# EPICS substitutions: iocCollimatorControl/R27CLM.substitutions
#BO,EPICS->PLC,Command
file "../../db/bo_word.template"{ pattern
{	P,		R,					PORT,		OFFSET,		MASK,		ZNAM,		ONAM	}
{	SR:R27:CLM:R27CLM:,	btn_LocalOrRemote,			R27CLM_BO1_Bits,	0,		0x0001,		Low,		High	}
{	SR:R27:CLM:R27CLM:,	btn_E_STOP,				R27CLM_BO1_Bits,	0,		0x0002,		Low,		High	}
{	SR:R27:CLM:R27CLM:,	m_restartTC,				R27CLM_BO1_Bits,	0,		0x0004,		Low,		High	}
{	SR:R27:CLM:R27CLM:,	btn_Move_Axis1,				R27CLM_BO2_Bits,	0,		0x0001,		Low,		High	}
{	SR:R27:CLM:R27CLM:,	btn_JogForward_Axis1,			R27CLM_BO2_Bits,	0,		0x0002,		Low,		High	}
{	SR:R27:CLM:R27CLM:,	btn_JogBackward_Axis1,			R27CLM_BO2_Bits,	0,		0x0004,		Low,		High	}
{	SR:R27:CLM:R27CLM:,	btn_Stop_Axis1,				R27CLM_BO2_Bits,	0,		0x0008,		Low,		High	}
{	SR:R27:CLM:R27CLM:,	btn_Reset_Axis1,			R27CLM_BO2_Bits,	0,		0x0010,		Low,		High	}
{	SR:R27:CLM:R27CLM:,	btn_SetPosition_Axis1,			R27CLM_BO2_Bits,	0,		0x0020,		Low,		High	}
{	SR:R27:CLM:R27CLM:,	LVDT1_FunctionOn,			R27CLM_BO2_Bits,	0,		0x0040,		Low,		High	}
{	SR:R27:CLM:R27CLM:,	LVDT1_ManualReleaseAlarm,		R27CLM_BO2_Bits,	0,		0x0080,		Low,		High	}
{	SR:R27:CLM:R27CLM:,	btn_Move_Axis2,				R27CLM_BO3_Bits,	0,		0x0001,		Low,		High	}
{	SR:R27:CLM:R27CLM:,	btn_JogForward_Axis2,			R27CLM_BO3_Bits,	0,		0x0002,		Low,		High	}
{	SR:R27:CLM:R27CLM:,	btn_JogBackward_Axis2,			R27CLM_BO3_Bits,	0,		0x0004,		Low,		High	}
{	SR:R27:CLM:R27CLM:,	btn_Stop_Axis2,				R27CLM_BO3_Bits,	0,		0x0008,		Low,		High	}
{	SR:R27:CLM:R27CLM:,	btn_Reset_Axis2,			R27CLM_BO3_Bits,	0,		0x0010,		Low,		High	}
{	SR:R27:CLM:R27CLM:,	btn_SetPosition_Axis2,			R27CLM_BO3_Bits,	0,		0x0020,		Low,		High	}
{	SR:R27:CLM:R27CLM:,	LVDT2_FunctionOn,			R27CLM_BO3_Bits,	0,		0x0040,		Low,		High	}
{	SR:R27:CLM:R27CLM:,	LVDT2_ManualReleaseAlarm,		R27CLM_BO3_Bits,	0,		0x0080,		Low,		High	}
{	SR:R27:CLM:R27CLM:,	btn_Move_AxisAll,			R27CLM_BO4_Bits,	0,		0x0001,		Low,		High	}
{	SR:R27:CLM:R27CLM:,	btn_JogForward_AxisAll,			R27CLM_BO4_Bits,	0,		0x0002,		Low,		High	}
{	SR:R27:CLM:R27CLM:,	btn_JogBackward_AxisAll,		R27CLM_BO4_Bits,	0,		0x0004,		Low,		High	}
{	SR:R27:CLM:R27CLM:,	btn_Stop_AxisAll,			R27CLM_BO4_Bits,	0,		0x0008,		Low,		High	}
{	SR:R27:CLM:R27CLM:,	btn_Reset_AxisAll,			R27CLM_BO4_Bits,	0,		0x0010,		Low,		High	}
}
#AO,EPICS->PLC,Command
file "../../db/aoFloat64.template" { pattern
{	P,           	R,               			PORT,      	OFFSET,   	DATA_TYPE,    	LOPR, 	HOPR, PREC	}
{	SR:R27:CLM:R27CLM:,	targetPositionAxis1,			R27CLM_AO1_FLOAT,	0,		FLOAT32_LE,	-1e6,	1e6,	4	}
{	SR:R27:CLM:R27CLM:,	targetVelocityAxis1,			R27CLM_AO1_FLOAT,	2,		FLOAT32_LE,	-1e6,	1e6,	4	}
{	SR:R27:CLM:R27CLM:,	increaseJogPositionAxis1,		R27CLM_AO1_FLOAT,	4,		FLOAT32_LE,	-1e6,	1e6,	4	}
{	SR:R27:CLM:R27CLM:,	Axis1_minPosition,			R27CLM_AO1_FLOAT,	6,		FLOAT32_LE,	-1e6,	1e6,	4	}
{	SR:R27:CLM:R27CLM:,	Axis1_maxPosition,			R27CLM_AO1_FLOAT,	8,		FLOAT32_LE,	-1e6,	1e6,	4	}
{	SR:R27:CLM:R27CLM:,	LVDT1_Threshold,			R27CLM_AO1_FLOAT,	10,		FLOAT32_LE,	-1e6,	1e6,	4	}
{	SR:R27:CLM:R27CLM:,	PositionSetValue_Axis1,			R27CLM_AO1_FLOAT,	12,		FLOAT32_LE,	-1e6,	1e6,	4	}
{	SR:R27:CLM:R27CLM:,	targetPositionAxis2,			R27CLM_AO2_FLOAT,	0,		FLOAT32_LE,	-1e6,	1e6,	4	}
{	SR:R27:CLM:R27CLM:,	targetVelocityAxis2,			R27CLM_AO2_FLOAT,	2,		FLOAT32_LE,	-1e6,	1e6,	4	}
{	SR:R27:CLM:R27CLM:,	increaseJogPositionAxis2,		R27CLM_AO2_FLOAT,	4,		FLOAT32_LE,	-1e6,	1e6,	4	}
{	SR:R27:CLM:R27CLM:,	Axis2_minPosition,			R27CLM_AO2_FLOAT,	6,		FLOAT32_LE,	-1e6,	1e6,	4	}
{	SR:R27:CLM:R27CLM:,	Axis2_maxPosition,			R27CLM_AO2_FLOAT,	8,		FLOAT32_LE,	-1e6,	1e6,	4	}
{	SR:R27:CLM:R27CLM:,	LVDT2_Threshold,			R27CLM_AO2_FLOAT,	10,		FLOAT32_LE,	-1e6,	1e6,	4	}
{	SR:R27:CLM:R27CLM:,	PositionSetValue_Axis2,			R27CLM_AO2_FLOAT,	12,		FLOAT32_LE,	-1e6,	1e6,	4	}
}
#R27CLM_BI,PLC->EPICS,Respond
file "../../db/bi_word.template"{ pattern
{	P,		R,					PORT,		OFFSET,		MASK,		ZNAM,		ONAM,		ZSV,		OSV,		SCAN		}
{	SR:R27:CLM:R27CLM:,	E_STOP_led,				R27CLM_BI1_Bits,	0,		0x0001,		Low,		High,		NO_ALARM,	NO_ALARM,	"I/O Intr"	}
{	SR:R27:CLM:R27CLM:,	Local_led,				R27CLM_BI1_Bits,	0,		0x0002,		Low,		High,		NO_ALARM,	NO_ALARM,	"I/O Intr"	}
{	SR:R27:CLM:R27CLM:,	Remote_led,				R27CLM_BI1_Bits,	0,		0x0004,		Low,		High,		NO_ALARM,	NO_ALARM,	"I/O Intr"	}
{	SR:R27:CLM:R27CLM:,	Error_led,				R27CLM_BI1_Bits,	0,		0x0008,		Low,		High,		NO_ALARM,	NO_ALARM,	"I/O Intr"	}
{	SR:R27:CLM:R27CLM:,	Axis1_error,				R27CLM_BI2_Bits,	0,		0x0001,		Low,		High,		NO_ALARM,	NO_ALARM,	"I/O Intr"	}
{	SR:R27:CLM:R27CLM:,	Axis1_moving,				R27CLM_BI2_Bits,	0,		0x0002,		Low,		High,		NO_ALARM,	NO_ALARM,	"I/O Intr"	}
{	SR:R27:CLM:R27CLM:,	foreward_limit_axis1,			R27CLM_BI2_Bits,	0,		0x0004,		Low,		High,		NO_ALARM,	NO_ALARM,	"I/O Intr"	}
{	SR:R27:CLM:R27CLM:,	backward_limit_axis1,			R27CLM_BI2_Bits,	0,		0x0008,		Low,		High,		NO_ALARM,	NO_ALARM,	"I/O Intr"	}
{	SR:R27:CLM:R27CLM:,	Moving_done_Axis1,			R27CLM_BI2_Bits,	0,		0x0010,		Low,		High,		NO_ALARM,	NO_ALARM,	"I/O Intr"	}
{	SR:R27:CLM:R27CLM:,	PositionSetDone_Axis1,			R27CLM_BI2_Bits,	0,		0x0020,		Low,		High,		NO_ALARM,	NO_ALARM,	"I/O Intr"	}
{	SR:R27:CLM:R27CLM:,	Axis2_error,				R27CLM_BI3_Bits,	0,		0x0001,		Low,		High,		NO_ALARM,	NO_ALARM,	"I/O Intr"	}
{	SR:R27:CLM:R27CLM:,	Axis2_moving,				R27CLM_BI3_Bits,	0,		0x0002,		Low,		High,		NO_ALARM,	NO_ALARM,	"I/O Intr"	}
{	SR:R27:CLM:R27CLM:,	foreward_limit_axis2,			R27CLM_BI3_Bits,	0,		0x0004,		Low,		High,		NO_ALARM,	NO_ALARM,	"I/O Intr"	}
{	SR:R27:CLM:R27CLM:,	backward_limit_axis2,			R27CLM_BI3_Bits,	0,		0x0008,		Low,		High,		NO_ALARM,	NO_ALARM,	"I/O Intr"	}
{	SR:R27:CLM:R27CLM:,	Moving_done_Axis2,			R27CLM_BI3_Bits,	0,		0x0010,		Low,		High,		NO_ALARM,	NO_ALARM,	"I/O Intr"	}
{	SR:R27:CLM:R27CLM:,	PositionSetDone_Axis2,			R27CLM_BI3_Bits,	0,		0x0020,		Low,		High,		NO_ALARM,	NO_ALARM,	"I/O Intr"	}
}
#R27CLM_AI,PLC->EPICS,Respond
file "../../db/aiFloat64.template"{ pattern
{	P,			R,					PORT,		OFFSET,		DATA_TYPE,	LOPR,	HOPR,	PREC,	SCAN			}
{	SR:R27:CLM:R27CLM:,	Axis1_Currentvelocity,			R27CLM_AI1_FLOAT,	0,		FLOAT32_LE,	-1e6,	1e6,	4,	"I/O Intr"		}
{	SR:R27:CLM:R27CLM:,	Axis1_CurrentPosition,			R27CLM_AI1_FLOAT,	2,		FLOAT32_LE,	-1e6,	1e6,	4,	"I/O Intr"		}
{	SR:R27:CLM:R27CLM:,	LVDT1_PV,				R27CLM_AI1_FLOAT,	4,		FLOAT32_LE,	-1e6,	1e6,	4,	"I/O Intr"		}
{	SR:R27:CLM:R27CLM:,	Axis2_Currentvelocity,			R27CLM_AI2_FLOAT,	0,		FLOAT32_LE,	-1e6,	1e6,	4,	"I/O Intr"		}
{	SR:R27:CLM:R27CLM:,	Axis2_CurrentPosition,			R27CLM_AI2_FLOAT,	2,		FLOAT32_LE,	-1e6,	1e6,	4,	"I/O Intr"		}
{	SR:R27:CLM:R27CLM:,	LVDT2_PV,				R27CLM_AI2_FLOAT,	4,		FLOAT32_LE,	-1e6,	1e6,	4,	"I/O Intr"		}
}
#Intin,PLC->EPICS,Respond
file "../../db/int64in.template"{ pattern
{	P,			R,			PORT,		OFFSET,		DATA_TYPE,	SCAN			}
{	SR:R27:CLM:R27CLM:,	ErrorId,		R27CLM_Intin,		0,		INT32_LE,	"I/O Intr"		}
}
#StringIn,PLC->EPICS,Respond
file "../../db/stringin.template"{ pattern
{	P,			R,				PORT,		OFFSET,		DATA_TYPE,	SCAN			}
{	SR:R27:CLM:R27CLM:,	ErrorDescription,		R27CLM_Stringin,	0,		STRING_LOW_HIGH,		"I/O Intr"		}
}
